GLOBALCONSTANTS DefaultPool_DIDO_Numeric (* Numeric object pool constants (ID, Scale, Offset, Decimals) *)
  PACKAGE Uebungen::const::UT::DIDO;
  VAR_GLOBAL CONSTANT
    OutputNumber_12000_N : logiBUS::utils::conversion::phys::NumericObjectPool_S := (u16ObjId := 12000, r32Scale := 1.0, i32Offset := 0, u8Decimals := 0);
    OutputNumber_12001_N : logiBUS::utils::conversion::phys::NumericObjectPool_S := (u16ObjId := 12001, r32Scale := 1.0, i32Offset := 0, u8Decimals := 0);
    OutputNumber_12002_N : logiBUS::utils::conversion::phys::NumericObjectPool_S := (u16ObjId := 12002, r32Scale := 1.0, i32Offset := 0, u8Decimals := 0);
    OutputNumber_12003_N : logiBUS::utils::conversion::phys::NumericObjectPool_S := (u16ObjId := 12003, r32Scale := 1.0, i32Offset := 0, u8Decimals := 0);
    OutputNumber_12004_N : logiBUS::utils::conversion::phys::NumericObjectPool_S := (u16ObjId := 12004, r32Scale := 1.0, i32Offset := 0, u8Decimals := 0);
    OutputNumber_12005_N : logiBUS::utils::conversion::phys::NumericObjectPool_S := (u16ObjId := 12005, r32Scale := 1.0, i32Offset := 0, u8Decimals := 0);
    OutputNumber_12006_N : logiBUS::utils::conversion::phys::NumericObjectPool_S := (u16ObjId := 12006, r32Scale := 1.0, i32Offset := 0, u8Decimals := 0);
    OutputNumber_12007_N : logiBUS::utils::conversion::phys::NumericObjectPool_S := (u16ObjId := 12007, r32Scale := 1.0, i32Offset := 0, u8Decimals := 0);
    OutputNumber_12008_N : logiBUS::utils::conversion::phys::NumericObjectPool_S := (u16ObjId := 12008, r32Scale := 1.0, i32Offset := 0, u8Decimals := 0);
    OutputNumber_12009_N : logiBUS::utils::conversion::phys::NumericObjectPool_S := (u16ObjId := 12009, r32Scale := 1.0, i32Offset := 0, u8Decimals := 0);
    OutputNumber_12010_N : logiBUS::utils::conversion::phys::NumericObjectPool_S := (u16ObjId := 12010, r32Scale := 1.0, i32Offset := 0, u8Decimals := 0);
    OutputNumber_12011_N : logiBUS::utils::conversion::phys::NumericObjectPool_S := (u16ObjId := 12011, r32Scale := 1.0, i32Offset := 0, u8Decimals := 0);
    OutputNumber_12012_N : logiBUS::utils::conversion::phys::NumericObjectPool_S := (u16ObjId := 12012, r32Scale := 1.0, i32Offset := 0, u8Decimals := 0);
    OutputNumber_12013_N : logiBUS::utils::conversion::phys::NumericObjectPool_S := (u16ObjId := 12013, r32Scale := 1.0, i32Offset := 0, u8Decimals := 0);
    OutputNumber_12014_N : logiBUS::utils::conversion::phys::NumericObjectPool_S := (u16ObjId := 12014, r32Scale := 1.0, i32Offset := 0, u8Decimals := 0);
    OutputNumber_12015_N : logiBUS::utils::conversion::phys::NumericObjectPool_S := (u16ObjId := 12015, r32Scale := 1.0, i32Offset := 0, u8Decimals := 0);
    OutputNumber_12016_N : logiBUS::utils::conversion::phys::NumericObjectPool_S := (u16ObjId := 12016, r32Scale := 1.0, i32Offset := 0, u8Decimals := 0);
    OutputNumber_12017_N : logiBUS::utils::conversion::phys::NumericObjectPool_S := (u16ObjId := 12017, r32Scale := 1.0, i32Offset := 0, u8Decimals := 0);
    OutputNumber_12018_N : logiBUS::utils::conversion::phys::NumericObjectPool_S := (u16ObjId := 12018, r32Scale := 1.0, i32Offset := 0, u8Decimals := 0);
    OutputNumber_12019_N : logiBUS::utils::conversion::phys::NumericObjectPool_S := (u16ObjId := 12019, r32Scale := 1.0, i32Offset := 0, u8Decimals := 0);
    OutputNumber_Tick_N : logiBUS::utils::conversion::phys::NumericObjectPool_S := (u16ObjId := 12020, r32Scale := 1.0, i32Offset := 0, u8Decimals := 0);
  END_VAR
END_GLOBALCONSTANTS
